FUNCTION_BLOCK ABSTRACT FB_Universal_FIFO IMPLEMENTS I_Universal_FIFO

VAR PERSISTENT    
	//Queue : ARRAY[0..MaxQueueSize-1] OF REAL;  // FIFO queue (size is 100 elements)
    Head : UINT := 0;  // Points to the next position to store data
    Tail : UINT := 0;  // Points to the oldest data position
    Count : UINT := 0;  // Number of elements currently in the FIFO
	bDataReady : BOOL; 
	eState : UINT;
END_VAR

VAR CONSTANT
	MaxQueueSize : UINT := 255;  // Number of elements in the FIFO queue

END_VAR

VAR_OUTPUT

   
END_VAR

PROPERTY CurrentCount : Uint
GET
CurrentCount := Count;
END_GET
END_PROPERTY

PROPERTY DataReady : BOOL
GET
DataReady := bDataReady;
END_GET
END_PROPERTY

PROPERTY HeadIndex : UINT
GET
HeadIndex := Head;
END_GET
END_PROPERTY

PROPERTY IsEmpty : bool
GET
IF Count = 0 THEN
	IsEmpty := TRUE;
ELSE
	IsEmpty := false;
END_IF
END_GET
END_PROPERTY

PROPERTY IsFull : bool
GET
IF count = MaxQueueSize THEN
	IsFull := TRUE;
ELSE 
	IsFull := FALSE;
END_IF
END_GET
END_PROPERTY

// if dataready return true, else return false// need overiding a part
METHOD MR_AckGetValue : BOOL
VAR_INPUT
END_VAR
IF bDataReady THEN
      
            // Data has been processed, so move to the next item in the queue
            Tail := (Tail + 1) MOD MaxQueueSize;
            Count := Count - 1;
            IF Count = 0 THEN
                bDataReady := FALSE;  // No more data to process
            END_IF
        
            // Data is still ready to be processed
        
    MR_AckGetValue := TRUE;   
ELSE 
	MR_AckGetValue := FALSE;
END_IF
// set oldest value in child fb here
// OldestData :=   Queue[Tail];
/////
END_METHOD

// need overide to reset oldestValue
METHOD MR_Reset : BOOL
VAR_INPUT
END_VAR
     Head := 0;
     Tail := 0;
     Count := 0;
	 bDataReady := FALSE;
	 MR_Reset := TRUE;
END_METHOD

PROPERTY TailIndex : Uint
GET
TailIndex := Tail;
END_GET
END_PROPERTY

END_FUNCTION_BLOCK

(* stored: Version 1.1.0.1, ProductVersion 3.1.4024.12
   POU FB_Universal_FIFO: Id {131aa9e2-58e3-45de-aafa-ea99eafcfdb0}, SpecialFunc None
   Property CurrentCount: Id {b394aead-437b-43a8-b08f-ed22975a952f}
   Get Get: Id {ea42aa8e-2694-4103-b382-20de3bb066f5}
   Property DataReady: Id {31648805-78a8-42f8-84a1-e6c84cdcf3f4}
   Get Get: Id {3a5c60e9-e41f-42ac-85af-ff42bc97f69f}
   Property HeadIndex: Id {faa593cb-1d80-4bce-ba98-616aadf9d26e}
   Get Get: Id {af63df6c-26ce-49a6-84cc-3ba9e5d6a369}
   Property IsEmpty: Id {6ac4853d-dd4b-4eab-ae86-df148cbd7815}
   Get Get: Id {d3b4f330-ad27-4609-8b4b-bce8d522bd59}
   Property IsFull: Id {9929d9b6-0d6d-4373-a85e-ad81b1b563c1}
   Get Get: Id {de385dae-c82c-49f8-8b9e-9ac114441ac0}
   Method MR_AckGetValue: Id {34860b74-6277-47be-b023-8c9d2a9707a8}
   Method MR_Reset: Id {573b5c3c-996e-49af-bd97-5cdc29213ede}
   Property TailIndex: Id {80acb226-1208-4672-938b-cb34f2e530e6}
   Get Get: Id {e7da5146-61aa-4feb-8312-8b8046365c71} *)
